(*
	Object 6040h: Control word (DS402)
	
*)
{attribute 'pack_mode' := '0'}
TYPE ST_DS402_ControlWord :
STRUCT
	b0_SwitchOn 					: BIT;
	b1_EnableVoltage				: BIT;
	b2_QuickStop					: BIT;
	b3_EnableOperation				: BIT;
	b4_OperationModeSpecific		: BIT;
	b5_OperationModeSpecific		: BIT;
	b6_OperationModeSpecific		: BIT;
	b7_FaultReset					: BIT;
	b8_Reserved						: BIT;
	b9_Reserved						: BIT;
	b10_Reserved					: BIT;
	b11_Reserved					: BIT;
	b12_Reserved					: BIT;
	b13_Reserved					: BIT;
	b14_Reserved					: BIT;
	b15_Reserved					: BIT;
END_STRUCT
END_TYPE

(* stored: Version 1.1.0.1, ProductVersion 3.1.4024.12
   DUT ST_DS402_ControlWord: Id {b02c0f2d-f6f8-05a9-12ee-03474f550937} *)
